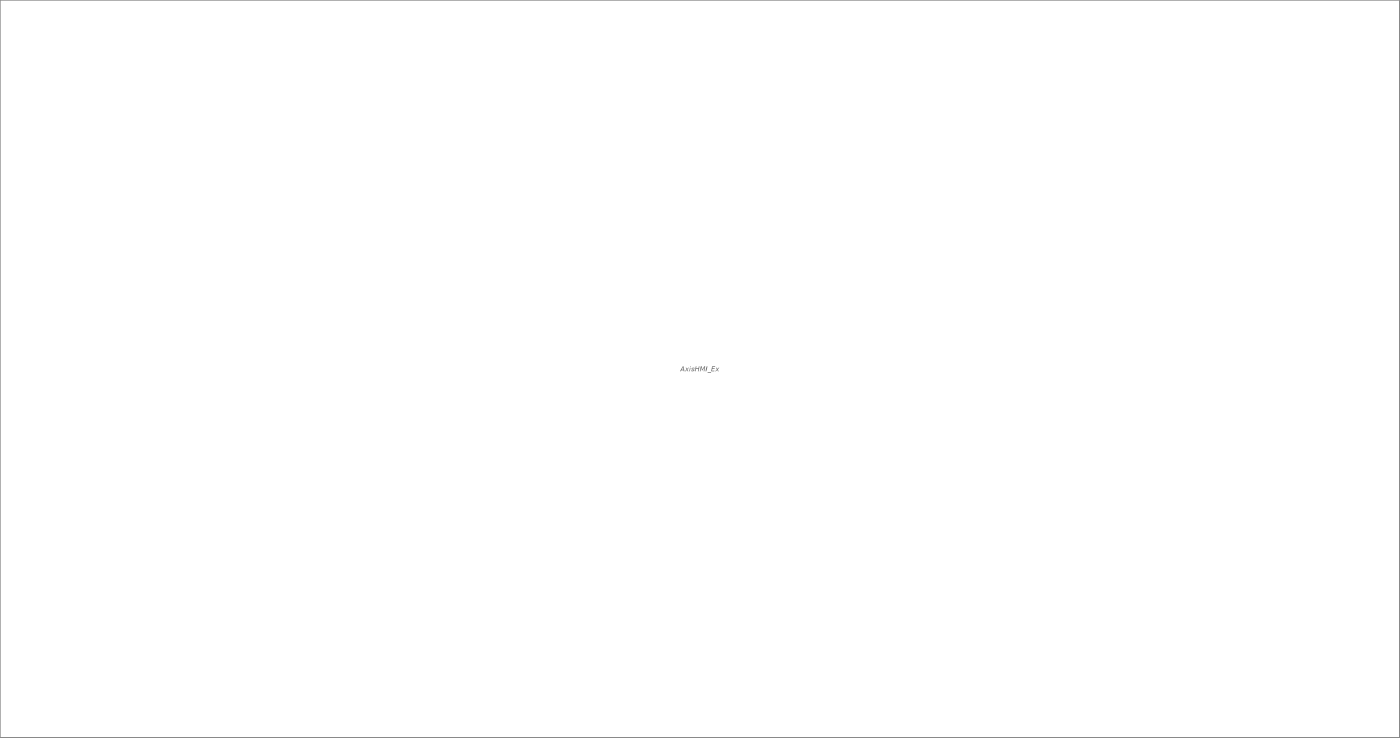
VISUALIZATION visu_ReM  // 2048x1080
    TabControl (0,0 2048x1080)
        shows AxisHMI_Ex(stAxisHMI := GVL.rem[G_HMI.iReM].lift[0].st_mcAxis, mcAxis := GVL.rem[G_HMI.iReM].lift[0].mcAxis, xError := GVL.rem[G_HMI.iReM].lift[0].mcAxis.xError)
        shows AxisHMI_Ex(stAxisHMI := GVL.rem[G_HMI.iReM].lift[1].st_mcAxis, mcAxis := GVL.rem[G_HMI.iReM].lift[1].mcAxis, xError := GVL.rem[G_HMI.iReM].lift[1].mcAxis.xError)
        shows v_rem_0(dIO_ReM := GVL.rem[G_HMI.iReM])
        shows v_rem_1(dIO_ReM := GVL.rem[G_HMI.iReM])
        shows Axis_HMI(st_axis_HMI := st_mcAxis[EN_Axis.Grip_axis])
        [0]: TabTitle=Lift0
        [1]: TabTitle=Lift1
        [2]: TabTitle=ReMIO_0, AxisHMI=gantrybase.st_mcAxis[EN_Axis.Z], mcAxis=gantrybase.mcAxis[EN_Axis.Z], Error=gantrybase.mcAxis[EN_Axis.Z].xError
        [3]: TabTitle=ReMIO_1
        [6]: TabTitle=Gripper
        p699000190: gantrybase.st_mcAxis[EN_Axis.X]
        p2837713833: gantrybase.mcAxis[EN_Axis.Z].sAxisName
        p520277221: gantrybase.mcAxis[EN_Axis.X].xError
        p3331604638: gantrybase.st_mcAxis[EN_Axis.Z]
        p1813558639: gantrybase.mcAxis[EN_Axis.Z].xError
        p1563495665: gantrybase.st_mcAxis[EN_Axis.Y]
        p2070126892: gantrybase.mcAxis[EN_Axis.Y].xError
        p3435970784: gantrybase.mcAxis[EN_Axis.X]
        p2829954345: gantrybase.mcAxis[EN_Axis.Y]
        p3218520426: gantrybase.mcAxis[EN_Axis.Z]
END_VISUALIZATION

(* stored: Version 1.1.0.1, ProductVersion 3.1.4024.12
   Visu visu_ReM: Id {4237067d-ba12-473e-bb87-3d8ec82551ac} *)
